Staubli VAL3: QueueFuncs.dtx


